(* Schneider Machine Expert - Basic project es2.1_2pompe_2max_3soglie_alternanza_giornaliera_con_minor_numero_ore, file version 3.0.0.0 *)
(* ProjectInformations: Name=New project *)

HARDWARE
  Cpu 0: TM221C40R
  EthernetConfiguration: NetworkName=M221, IpAllocationMode=FixedAddress, IpAddress=0.0.0.0, SubnetMask=0.0.0.0
  SerialLineConfiguration: Baud=Baud19200, Parity=ParityEven, DataBits=DataBits8, StopBits=StopBits1, PhysicalMedium=PhysicalMediumRs485, TransmissionMode=TransmissionModeModbusRtu, SlaveId=1, Addressing=SlaveAddressing
  MastTask: UsePeriodScanMode=false, PeriodScan=100
  FastTask: Period=255
  CpuBehavior: StartingMode=StartAsPreviousState, AutoSaveRamOnEeprom=true, WatchdogPeriod=250

SYMBOLS  (address, symbol, comment, settings)
  %M0       P1_USABILE
  %M1       P2_USABILE
  %M2       P1_COMANDATA  "Stesso valore di P1_CMD. Permette di identificare gli edges, visto che P1_CMD non può farlo."
  %M3       P2_COMANDATA  "Stesso valore di P2_CMD. Permette di identificare gli edges, visto che P2_CMD non può farlo."
  %M4       P3_USABILE
  %M5       P4_USABILE
  %M6       P3_COMANDATA
  %M7       P4_COMANDATA
  %M8       ESISTE_PROX_POMPA_CON_MINOR_ORE  "Nel loop, può non esistere una prossima pompa usabile e non comandata con il minor numero ore."
  %M9       ORA_E_00  "E' mezzanotte?"
  %M10      DECISO_ORDINE  "In intervallo in cui alternare le pompe per altern. giorn., è stata deciso quale sarà prossima pompa con minor ore?"
  %M11      PRIMA_POMPA_COMANDATA  "La prima pompa dell'ordine è stata effettivamente comandata quando serviva?"
  %M12      SECONDA_POMPA_COMANDATA  "La seconda pompa dell'ordine è stata effettivamente comandata quando serviva?"
  %S6       SB_TB1S  "Time base of 1 s generated by an internal clock"
  %SW51     SW_RTCHHMM  "RTC Function: contains in BCD HHMM: hour and minute"
  %MW0      NUM_POMPE_DA_COMANDARE  "Numero di pompe da comandare in base alle soglie raggiunte."
  %MW1      NUM_POMPE_COMANDATE  "Numero di pompe effettivamente comandate, in base alle loro disponibilità."
  %MW2      NUM_POMPE  "Numero di pompe totali."
  %MW3      ULTIMO_MINOR_SECONDI_LAVORATI  "Ultimi secondi lavorati più piccoli (valore temporaneo, da usare solo nel loop)."
  %MW4      PROSSIMA_POMPA_DA_COMANDARE  "Numero da 1 a NUM_POMPE che indica la prossima pompa da comandare."
  %MW5      POMPA_ATTUALE_LOOP  "Pompa attuale nel loop."
  %MW6      NUM_POMPE_COMANDATE_MAX  "Num"
  %MW7      CONTA_POMPE_COMANDATE_MAX  "Da usare in loop e da resettare.  Assume il valore da 1 fino a NUM_POMPE_COMANDATE_MAX."
  %MW8      ORDINE_PRIMA_POMPA
  %MW9      ORDINE_SECONDA_POMPA
  %MW10     ORDINE_TERZA_POMPA
  %MW11     ORDINE_QUARTA_POMPA
  %C0       CONTATORE_P1_SECONDI_LAVORATI  [Preset=0]
  %C1       CONTATORE_P2_SECONDI_LAVORATI  [Preset=0]
  %C2       CONTATORE_P3_SECONDI_LAVORATI  [Preset=0]
  %C3       CONTATORE_P4_SECONDI_LAVORATI  [Preset=0]
  %I0.0     P1_AUTO
  %I0.1     P1_MOTO
  %I0.2     P1_ANOMALIA
  %I0.3     P2_AUTO
  %I0.4     P2_MOTO
  %I0.5     P2_ANOMALIA
  %I0.6     LVL_MIN
  %I0.7     LVL_MAX1
  %I0.8     LVL_MAX2
  %I0.9     P3_AUTO
  %I0.10    P3_MOTO
  %I0.11    P3_ANOMALIA
  %I0.12    P4_AUTO
  %I0.13    P4_MOTO
  %I0.14    P4_ANOMALIA
  %I0.15    LVL_MAX3
  %Q0.0     P1_CMD
  %Q0.1     P2_CMD
  %Q0.2     P3_CMD
  %Q0.3     P4_CMD

POU New POU
  (* SectionNumber=1 *)

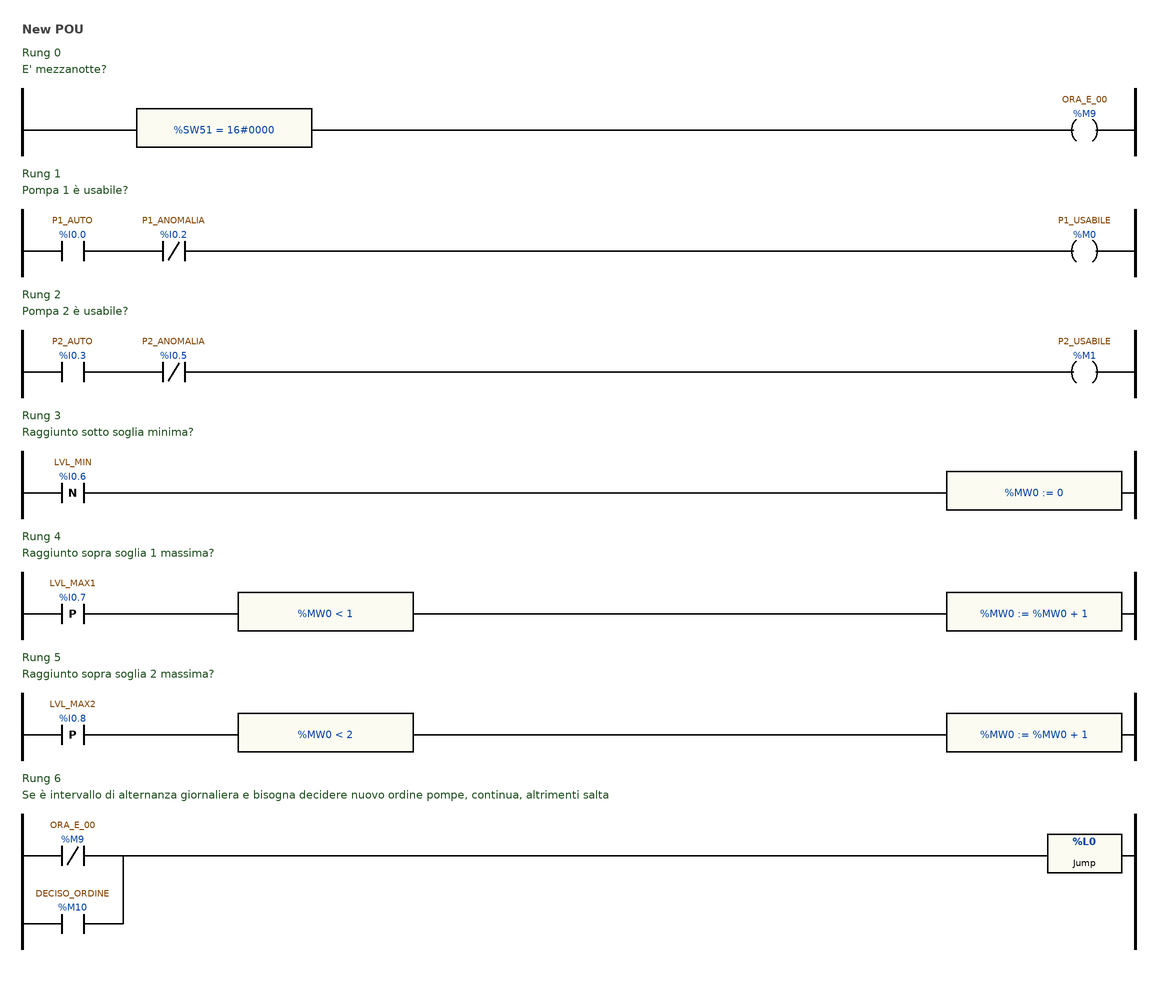

// Rung 0
// E' mezzanotte?
  LD [ %SW51 = 16#0000 ]  (* SW_RTCHHMM *)
  ST %M9                  (* ORA_E_00 *)
  // as ST:
  //   ORA_E_00 := SW_RTCHHMM = 16#0000;

// Rung 1
// Pompa 1 è usabile?
  LD %I0.0                (* P1_AUTO *)
  ANDN %I0.2              (* P1_ANOMALIA *)
  ST %M0                  (* P1_USABILE *)
  // as ST:
  //   P1_USABILE := P1_AUTO AND NOT P1_ANOMALIA;

// Rung 2
// Pompa 2 è usabile?
  LD %I0.3                (* P2_AUTO *)
  ANDN %I0.5              (* P2_ANOMALIA *)
  ST %M1                  (* P2_USABILE *)
  // as ST:
  //   P2_USABILE := P2_AUTO AND NOT P2_ANOMALIA;

// Rung 3
// Raggiunto sotto soglia minima?
  LDF %I0.6               (* LVL_MIN *)
  [ %MW0 := 0 ]           (* NUM_POMPE_DA_COMANDARE *)
  // as ST:
  //   IF FALLING(LVL_MIN) THEN NUM_POMPE_DA_COMANDARE := 0; END_IF;

// Rung 4
// Raggiunto sopra soglia 1 massima?
  LDR %I0.7               (* LVL_MAX1 *)
  AND [ %MW0 < 1 ]        (* NUM_POMPE_DA_COMANDARE *)
  [ %MW0 := %MW0 + 1 ]    (* NUM_POMPE_DA_COMANDARE, NUM_POMPE_DA_COMANDARE *)
  // as ST:
  //   IF RISING(LVL_MAX1) AND NUM_POMPE_DA_COMANDARE < 1 THEN NUM_POMPE_DA_COMANDARE := NUM_POMPE_DA_COMANDARE + 1; END_IF;

// Rung 5
// Raggiunto sopra soglia 2 massima?
  LDR %I0.8               (* LVL_MAX2 *)
  AND [ %MW0 < 2 ]        (* NUM_POMPE_DA_COMANDARE *)
  [ %MW0 := %MW0 + 1 ]    (* NUM_POMPE_DA_COMANDARE, NUM_POMPE_DA_COMANDARE *)
  // as ST:
  //   IF RISING(LVL_MAX2) AND NUM_POMPE_DA_COMANDARE < 2 THEN NUM_POMPE_DA_COMANDARE := NUM_POMPE_DA_COMANDARE + 1; END_IF;

// Rung 6
// Se è intervallo di alternanza giornaliera e bisogna decidere nuovo ordine pompe, continua, altrimenti salta
  LDN %M9                 (* ORA_E_00 *)
  OR %M10                 (* DECISO_ORDINE *)
  JMPC %L0
  // as ST:
  //   IF NOT ORA_E_00 OR DECISO_ORDINE THEN JMP %L0; END_IF;

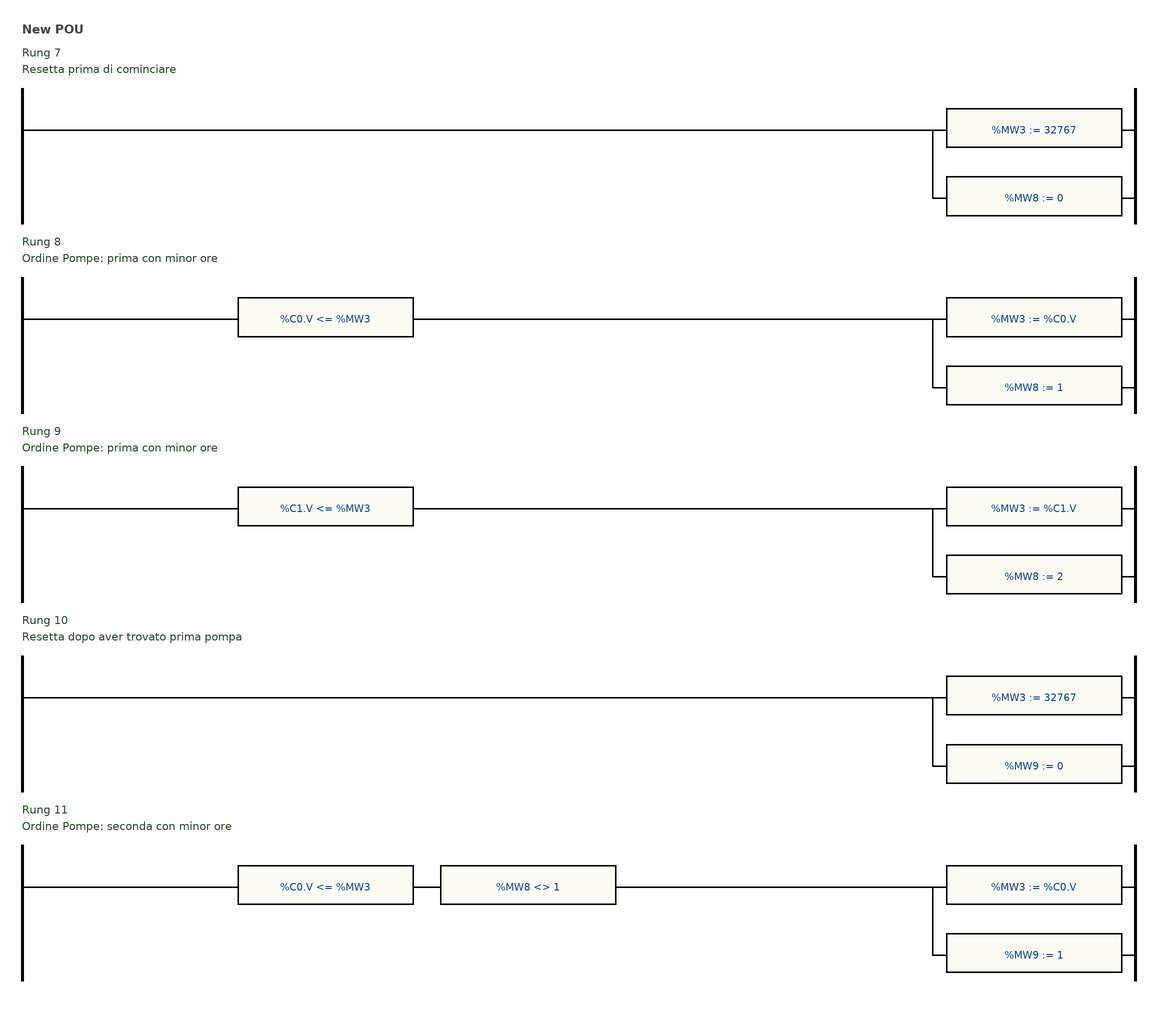

// Rung 7
// Resetta prima di cominciare
  LD 1
  [ %MW3 := 32767 ]       (* ULTIMO_MINOR_SECONDI_LAVORATI *)
  [ %MW8 := 0 ]           (* ORDINE_PRIMA_POMPA *)
  // as ST:
  //   ULTIMO_MINOR_SECONDI_LAVORATI := 32767;
  //   ORDINE_PRIMA_POMPA := 0;

// Rung 8
// Ordine Pompe: prima con minor ore
  LD [ %C0.V <= %MW3 ]    (* CONTATORE_P1_SECONDI_LAVORATI, ULTIMO_MINOR_SECONDI_LAVORATI *)
  [ %MW3 := %C0.V ]       (* ULTIMO_MINOR_SECONDI_LAVORATI, CONTATORE_P1_SECONDI_LAVORATI *)
  [ %MW8 := 1 ]           (* ORDINE_PRIMA_POMPA *)
  // as ST:
  //   _t1 := CONTATORE_P1_SECONDI_LAVORATI.V <= ULTIMO_MINOR_SECONDI_LAVORATI;
  //   IF _t1 THEN ULTIMO_MINOR_SECONDI_LAVORATI := CONTATORE_P1_SECONDI_LAVORATI.V; END_IF;
  //   IF _t1 THEN ORDINE_PRIMA_POMPA := 1; END_IF;

// Rung 9
// Ordine Pompe: prima con minor ore
  LD [ %C1.V <= %MW3 ]    (* CONTATORE_P2_SECONDI_LAVORATI, ULTIMO_MINOR_SECONDI_LAVORATI *)
  [ %MW3 := %C1.V ]       (* ULTIMO_MINOR_SECONDI_LAVORATI, CONTATORE_P2_SECONDI_LAVORATI *)
  [ %MW8 := 2 ]           (* ORDINE_PRIMA_POMPA *)
  // as ST:
  //   _t1 := CONTATORE_P2_SECONDI_LAVORATI.V <= ULTIMO_MINOR_SECONDI_LAVORATI;
  //   IF _t1 THEN ULTIMO_MINOR_SECONDI_LAVORATI := CONTATORE_P2_SECONDI_LAVORATI.V; END_IF;
  //   IF _t1 THEN ORDINE_PRIMA_POMPA := 2; END_IF;

// Rung 10
// Resetta dopo aver trovato prima pompa
  LD 1
  [ %MW3 := 32767 ]       (* ULTIMO_MINOR_SECONDI_LAVORATI *)
  [ %MW9 := 0 ]           (* ORDINE_SECONDA_POMPA *)
  // as ST:
  //   ULTIMO_MINOR_SECONDI_LAVORATI := 32767;
  //   ORDINE_SECONDA_POMPA := 0;

// Rung 11
// Ordine Pompe: seconda con minor ore
  LD [ %C0.V <= %MW3 ]    (* CONTATORE_P1_SECONDI_LAVORATI, ULTIMO_MINOR_SECONDI_LAVORATI *)
  AND [ %MW8 <> 1 ]       (* ORDINE_PRIMA_POMPA *)
  [ %MW3 := %C0.V ]       (* ULTIMO_MINOR_SECONDI_LAVORATI, CONTATORE_P1_SECONDI_LAVORATI *)
  [ %MW9 := 1 ]           (* ORDINE_SECONDA_POMPA *)
  // as ST:
  //   _t1 := CONTATORE_P1_SECONDI_LAVORATI.V <= ULTIMO_MINOR_SECONDI_LAVORATI AND ORDINE_PRIMA_POMPA <> 1;
  //   IF _t1 THEN ULTIMO_MINOR_SECONDI_LAVORATI := CONTATORE_P1_SECONDI_LAVORATI.V; END_IF;
  //   IF _t1 THEN ORDINE_SECONDA_POMPA := 1; END_IF;

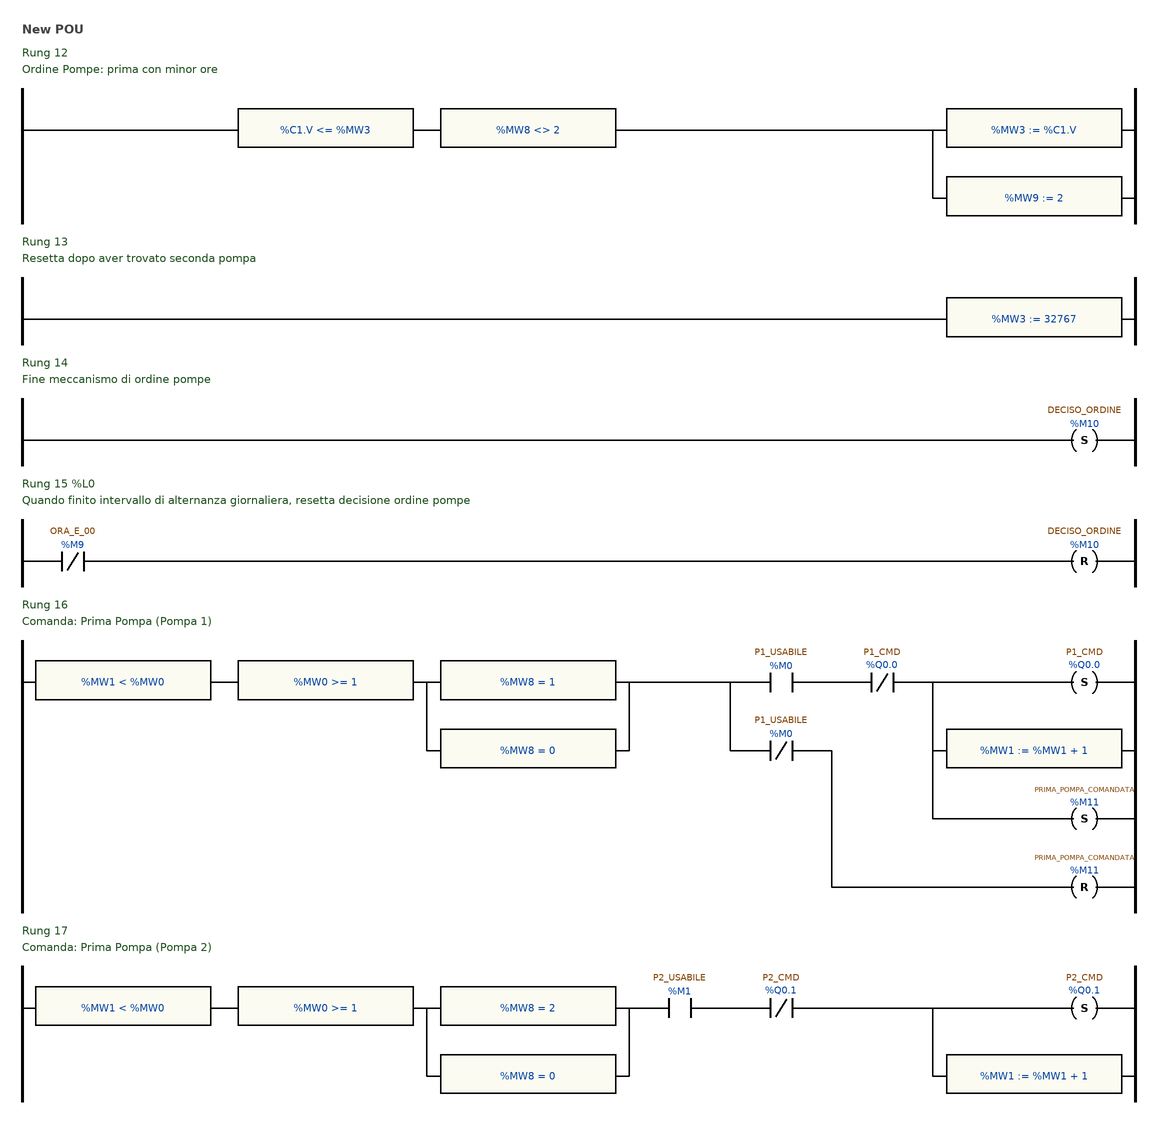

// Rung 12
// Ordine Pompe: prima con minor ore
  LD [ %C1.V <= %MW3 ]    (* CONTATORE_P2_SECONDI_LAVORATI, ULTIMO_MINOR_SECONDI_LAVORATI *)
  AND [ %MW8 <> 2 ]       (* ORDINE_PRIMA_POMPA *)
  [ %MW3 := %C1.V ]       (* ULTIMO_MINOR_SECONDI_LAVORATI, CONTATORE_P2_SECONDI_LAVORATI *)
  [ %MW9 := 2 ]           (* ORDINE_SECONDA_POMPA *)
  // as ST:
  //   _t1 := CONTATORE_P2_SECONDI_LAVORATI.V <= ULTIMO_MINOR_SECONDI_LAVORATI AND ORDINE_PRIMA_POMPA <> 2;
  //   IF _t1 THEN ULTIMO_MINOR_SECONDI_LAVORATI := CONTATORE_P2_SECONDI_LAVORATI.V; END_IF;
  //   IF _t1 THEN ORDINE_SECONDA_POMPA := 2; END_IF;

// Rung 13
// Resetta dopo aver trovato seconda pompa
  LD 1
  [ %MW3 := 32767 ]       (* ULTIMO_MINOR_SECONDI_LAVORATI *)
  // as ST:
  //   ULTIMO_MINOR_SECONDI_LAVORATI := 32767;

// Rung 14
// Fine meccanismo di ordine pompe
  LD 1
  S %M10                  (* DECISO_ORDINE *)
  // as ST:
  //   DECISO_ORDINE := TRUE;

// Rung 15 %L0
// Quando finito intervallo di alternanza giornaliera, resetta decisione ordine pompe
  %L0:
  LDN %M9                 (* ORA_E_00 *)
  R %M10                  (* DECISO_ORDINE *)
  // as ST:
  //   %L0:
  //   IF NOT ORA_E_00 THEN DECISO_ORDINE := FALSE; END_IF;

// Rung 16
// Comanda: Prima Pompa (Pompa 1)
  (* no IL stored for this rung *)

// Rung 17
// Comanda: Prima Pompa (Pompa 2)
  LD [ %MW1 < %MW0 ]      (* NUM_POMPE_COMANDATE, NUM_POMPE_DA_COMANDARE *)
  AND [ %MW0 >= 1 ]       (* NUM_POMPE_DA_COMANDARE *)
  AND( [ %MW8 = 2 ]       (* ORDINE_PRIMA_POMPA *)
  OR [ %MW8 = 0 ]         (* ORDINE_PRIMA_POMPA *)
  )
  AND %M1                 (* P2_USABILE *)
  ANDN %Q0.1              (* P2_CMD *)
  S %Q0.1                 (* P2_CMD *)
  [ %MW1 := %MW1 + 1 ]    (* NUM_POMPE_COMANDATE, NUM_POMPE_COMANDATE *)
  // as ST:
  //   _t1 := NUM_POMPE_COMANDATE < NUM_POMPE_DA_COMANDARE AND NUM_POMPE_DA_COMANDARE >= 1 AND (ORDINE_PRIMA_POMPA = 2 OR ORDINE_PRIMA_POMPA = 0) AND P2_USABILE AND NOT P2_CMD;
  //   IF _t1 THEN P2_CMD := TRUE; END_IF;
  //   IF _t1 THEN NUM_POMPE_COMANDATE := NUM_POMPE_COMANDATE + 1; END_IF;

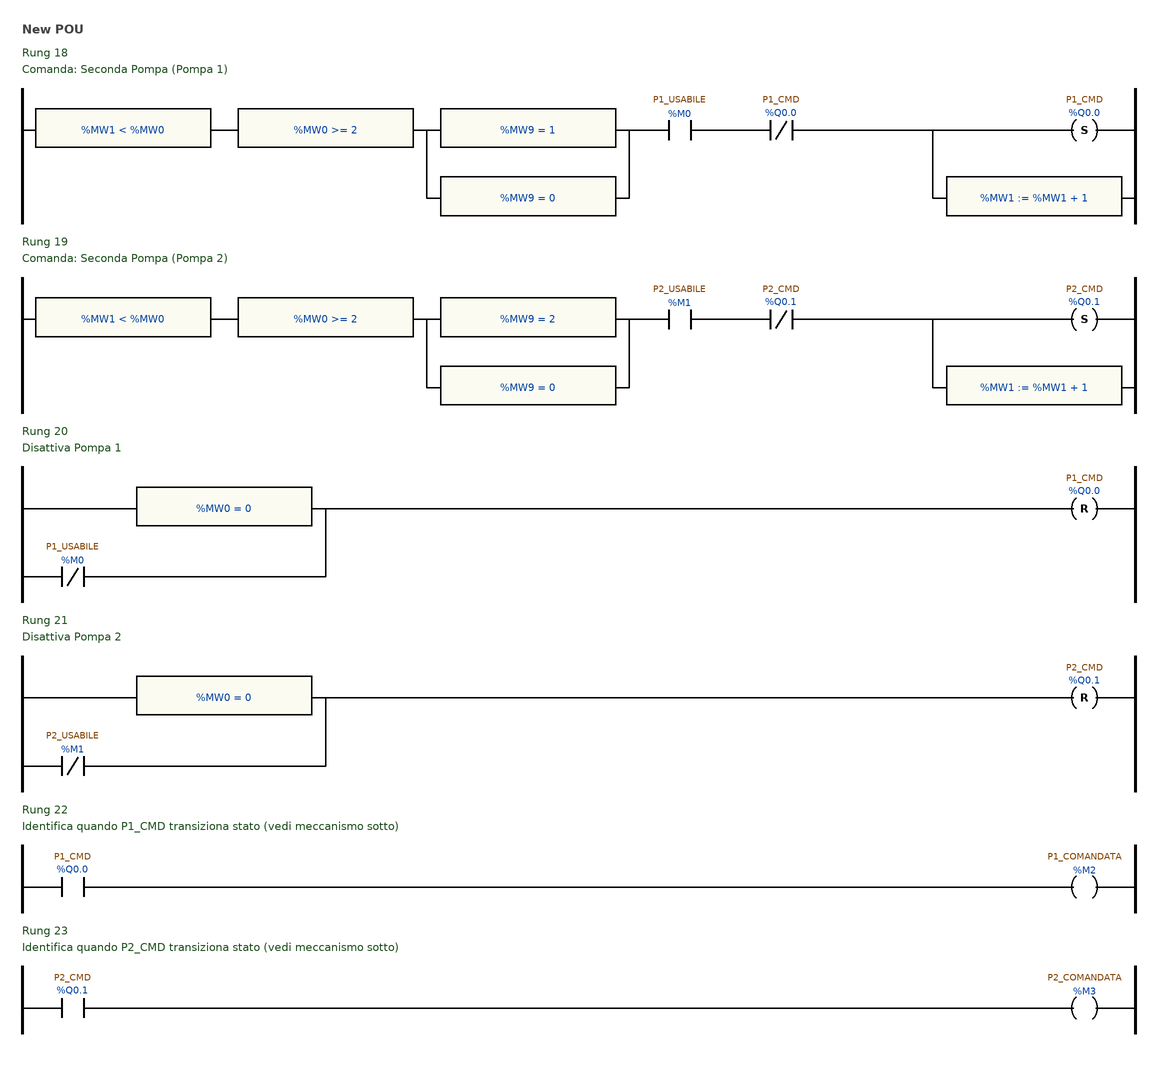

// Rung 18
// Comanda: Seconda Pompa (Pompa 1)
  LD [ %MW1 < %MW0 ]      (* NUM_POMPE_COMANDATE, NUM_POMPE_DA_COMANDARE *)
  AND [ %MW0 >= 2 ]       (* NUM_POMPE_DA_COMANDARE *)
  AND( [ %MW9 = 1 ]       (* ORDINE_SECONDA_POMPA *)
  OR [ %MW9 = 0 ]         (* ORDINE_SECONDA_POMPA *)
  )
  AND %M0                 (* P1_USABILE *)
  ANDN %Q0.0              (* P1_CMD *)
  S %Q0.0                 (* P1_CMD *)
  [ %MW1 := %MW1 + 1 ]    (* NUM_POMPE_COMANDATE, NUM_POMPE_COMANDATE *)
  // as ST:
  //   _t1 := NUM_POMPE_COMANDATE < NUM_POMPE_DA_COMANDARE AND NUM_POMPE_DA_COMANDARE >= 2 AND (ORDINE_SECONDA_POMPA = 1 OR ORDINE_SECONDA_POMPA = 0) AND P1_USABILE AND NOT P1_CMD;
  //   IF _t1 THEN P1_CMD := TRUE; END_IF;
  //   IF _t1 THEN NUM_POMPE_COMANDATE := NUM_POMPE_COMANDATE + 1; END_IF;

// Rung 19
// Comanda: Seconda Pompa (Pompa 2)
  LD [ %MW1 < %MW0 ]      (* NUM_POMPE_COMANDATE, NUM_POMPE_DA_COMANDARE *)
  AND [ %MW0 >= 2 ]       (* NUM_POMPE_DA_COMANDARE *)
  AND( [ %MW9 = 2 ]       (* ORDINE_SECONDA_POMPA *)
  OR [ %MW9 = 0 ]         (* ORDINE_SECONDA_POMPA *)
  )
  AND %M1                 (* P2_USABILE *)
  ANDN %Q0.1              (* P2_CMD *)
  S %Q0.1                 (* P2_CMD *)
  [ %MW1 := %MW1 + 1 ]    (* NUM_POMPE_COMANDATE, NUM_POMPE_COMANDATE *)
  // as ST:
  //   _t1 := NUM_POMPE_COMANDATE < NUM_POMPE_DA_COMANDARE AND NUM_POMPE_DA_COMANDARE >= 2 AND (ORDINE_SECONDA_POMPA = 2 OR ORDINE_SECONDA_POMPA = 0) AND P2_USABILE AND NOT P2_CMD;
  //   IF _t1 THEN P2_CMD := TRUE; END_IF;
  //   IF _t1 THEN NUM_POMPE_COMANDATE := NUM_POMPE_COMANDATE + 1; END_IF;

// Rung 20
// Disattiva Pompa 1
  LD [ %MW0 = 0 ]         (* NUM_POMPE_DA_COMANDARE *)
  ORN %M0                 (* P1_USABILE *)
  R %Q0.0                 (* P1_CMD *)
  // as ST:
  //   IF NUM_POMPE_DA_COMANDARE = 0 OR NOT P1_USABILE THEN P1_CMD := FALSE; END_IF;

// Rung 21
// Disattiva Pompa 2
  LD [ %MW0 = 0 ]         (* NUM_POMPE_DA_COMANDARE *)
  ORN %M1                 (* P2_USABILE *)
  R %Q0.1                 (* P2_CMD *)
  // as ST:
  //   IF NUM_POMPE_DA_COMANDARE = 0 OR NOT P2_USABILE THEN P2_CMD := FALSE; END_IF;

// Rung 22
// Identifica quando P1_CMD transiziona stato (vedi meccanismo sotto)
  LD %Q0.0                (* P1_CMD *)
  ST %M2                  (* P1_COMANDATA *)
  // as ST:
  //   P1_COMANDATA := P1_CMD;

// Rung 23
// Identifica quando P2_CMD transiziona stato (vedi meccanismo sotto)
  LD %Q0.1                (* P2_CMD *)
  ST %M3                  (* P2_COMANDATA *)
  // as ST:
  //   P2_COMANDATA := P2_CMD;

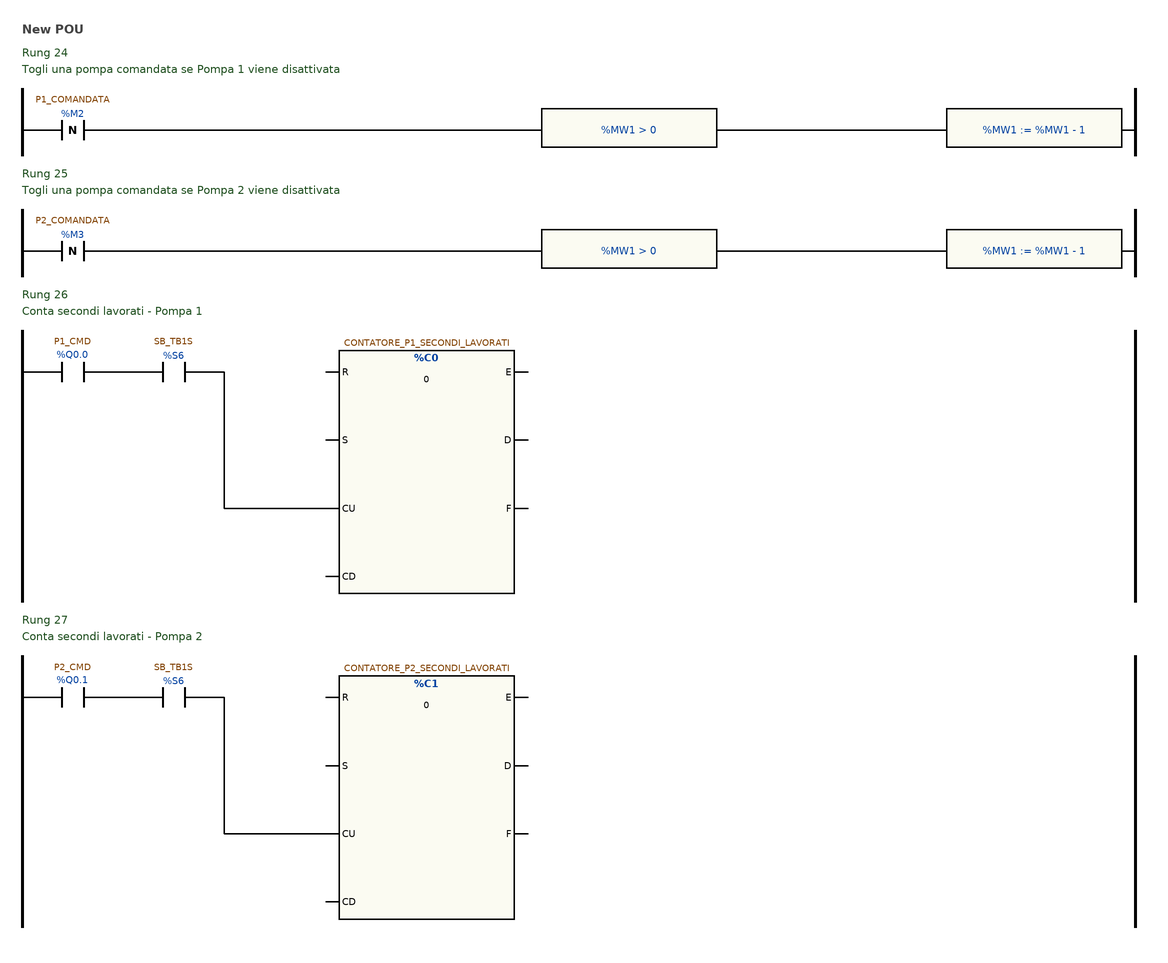

// Rung 24
// Togli una pompa comandata se Pompa 1 viene disattivata
  LDF %M2                 (* P1_COMANDATA *)
  AND [ %MW1 > 0 ]        (* NUM_POMPE_COMANDATE *)
  [ %MW1 := %MW1 - 1 ]    (* NUM_POMPE_COMANDATE, NUM_POMPE_COMANDATE *)
  // as ST:
  //   IF FALLING(P1_COMANDATA) AND NUM_POMPE_COMANDATE > 0 THEN NUM_POMPE_COMANDATE := NUM_POMPE_COMANDATE - 1; END_IF;

// Rung 25
// Togli una pompa comandata se Pompa 2 viene disattivata
  LDF %M3                 (* P2_COMANDATA *)
  AND [ %MW1 > 0 ]        (* NUM_POMPE_COMANDATE *)
  [ %MW1 := %MW1 - 1 ]    (* NUM_POMPE_COMANDATE, NUM_POMPE_COMANDATE *)
  // as ST:
  //   IF FALLING(P2_COMANDATA) AND NUM_POMPE_COMANDATE > 0 THEN NUM_POMPE_COMANDATE := NUM_POMPE_COMANDATE - 1; END_IF;

// Rung 26
// Conta secondi lavorati - Pompa 1
  BLK %C0                 (* CONTATORE_P1_SECONDI_LAVORATI *)
  LD %Q0.0                (* P1_CMD *)
  AND %S6                 (* SB_TB1S *)
  CU
  END_BLK
  // as ST:
  //   CONTATORE_P1_SECONDI_LAVORATI(CU := P1_CMD AND SB_TB1S);

// Rung 27
// Conta secondi lavorati - Pompa 2
  BLK %C1                 (* CONTATORE_P2_SECONDI_LAVORATI *)
  LD %Q0.1                (* P2_CMD *)
  AND %S6                 (* SB_TB1S *)
  CU
  END_BLK
  // as ST:
  //   CONTATORE_P2_SECONDI_LAVORATI(CU := P2_CMD AND SB_TB1S);
